// Mitsubishi GX Developer project: PLC_PCO520L2   PLC: Q06UDEH

PROGRAM MAIN
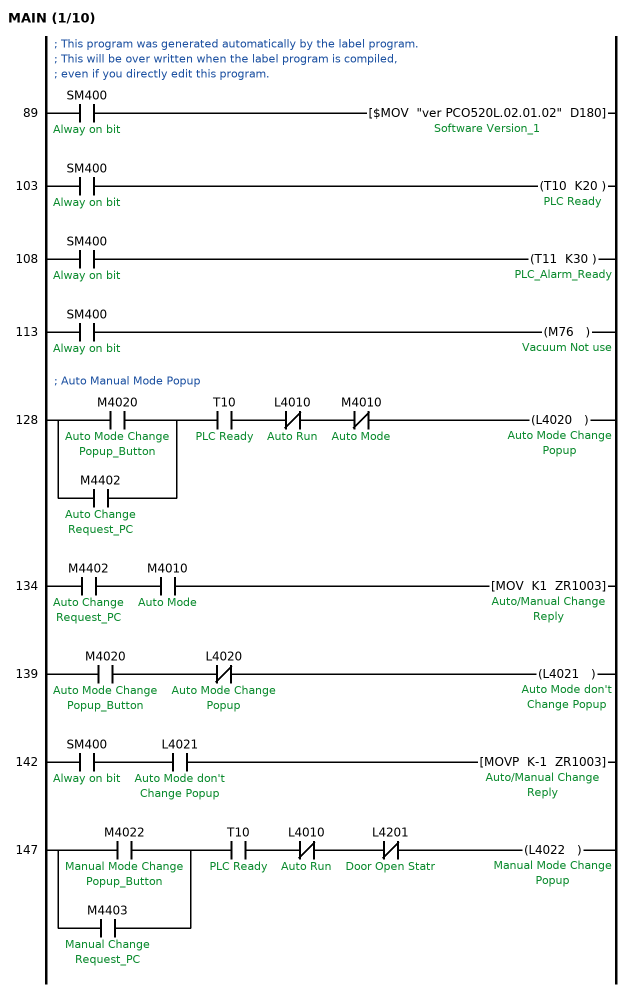
; This program was generated automatically by the label program.
; This will be over written when the label program is compiled,
; even if you directly edit this program.
89    LD      SM400  ; Alway on bit
      $MOV    "ver PCO520L.02.01.02" D180  ; Software Version_1
103   LD      SM400  ; Alway on bit
      OUT     T10 K20  ; PLC Ready
108   LD      SM400  ; Alway on bit
      OUT     T11 K30  ; PLC_Alarm_Ready
113   LD      SM400  ; Alway on bit
      OUT     M76  ; Vacuum Not use
; Auto Manual Mode Popup
128   LD      M4020  ; Auto Mode Change Popup_Button
      OR      M4402  ; Auto Change Request_PC
      AND     T10  ; PLC Ready
      ANI     L4010  ; Auto Run
      ANI     M4010  ; Auto Mode
      OUT     L4020  ; Auto Mode Change Popup
134   LD      M4402  ; Auto Change Request_PC
      AND     M4010  ; Auto Mode
      MOV     K1 ZR1003  ; Auto/Manual Change Reply
139   LD      M4020  ; Auto Mode Change Popup_Button
      ANI     L4020  ; Auto Mode Change Popup
      OUT     L4021  ; Auto Mode don't Change Popup
142   LD      SM400  ; Alway on bit
      AND     L4021  ; Auto Mode don't Change Popup
      MOVP    K-1 ZR1003
147   LD      M4022  ; Manual Mode Change Popup_Button
      OR      M4403  ; Manual Change Request_PC
      AND     T10  ; PLC Ready
      ANI     L4010  ; Auto Run
      ANI     L4201  ; Door Open Statr
      OUT     L4022  ; Manual Mode Change Popup
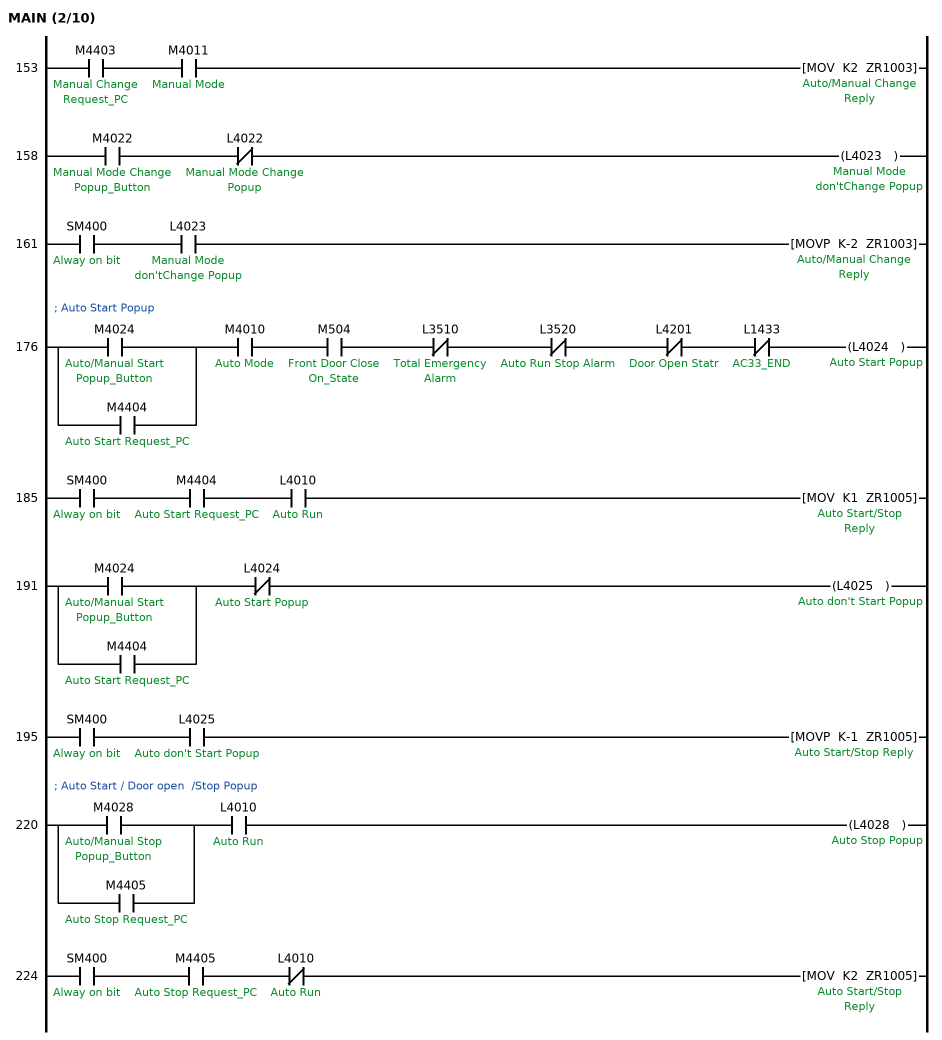
153   LD      M4403  ; Manual Change Request_PC
      AND     M4011  ; Manual Mode
      MOV     K2 ZR1003
158   LD      M4022  ; Manual Mode Change Popup_Button
      ANI     L4022  ; Manual Mode Change Popup
      OUT     L4023  ; Manual Mode  don'tChange Popup
161   LD      SM400  ; Alway on bit
      AND     L4023  ; Manual Mode  don'tChange Popup
      MOVP    K-2 ZR1003
; Auto Start Popup
176   LD      M4024  ; Auto/Manual Start Popup_Button
      OR      M4404  ; Auto Start Request_PC
      AND     M4010  ; Auto Mode
      AND     M504  ; Front Door Close On_State
      ANI     L3510  ; Total Emergency Alarm
      ANI     L3520  ; Auto Run Stop Alarm
      ANI     L4201  ; Door Open Statr
      ANI     L1433  ; AC33_END
      OUT     L4024  ; Auto Start Popup
185   LD      SM400  ; Alway on bit
      AND     M4404  ; Auto Start Request_PC
      AND     L4010  ; Auto Run
      MOV     K1 ZR1005  ; Auto Start/Stop Reply
191   LD      M4024  ; Auto/Manual Start Popup_Button
      OR      M4404  ; Auto Start Request_PC
      ANI     L4024  ; Auto Start Popup
      OUT     L4025  ; Auto don't Start Popup
195   LD      SM400  ; Alway on bit
      AND     L4025  ; Auto don't Start Popup
      MOVP    K-1 ZR1005
; Auto Start / Door open  /Stop Popup
220   LD      M4028  ; Auto/Manual Stop Popup_Button
      OR      M4405  ; Auto Stop Request_PC
      AND     L4010  ; Auto Run
      OUT     L4028  ; Auto Stop Popup
224   LD      SM400  ; Alway on bit
      AND     M4405  ; Auto Stop Request_PC
      ANI     L4010  ; Auto Run
      MOV     K2 ZR1005
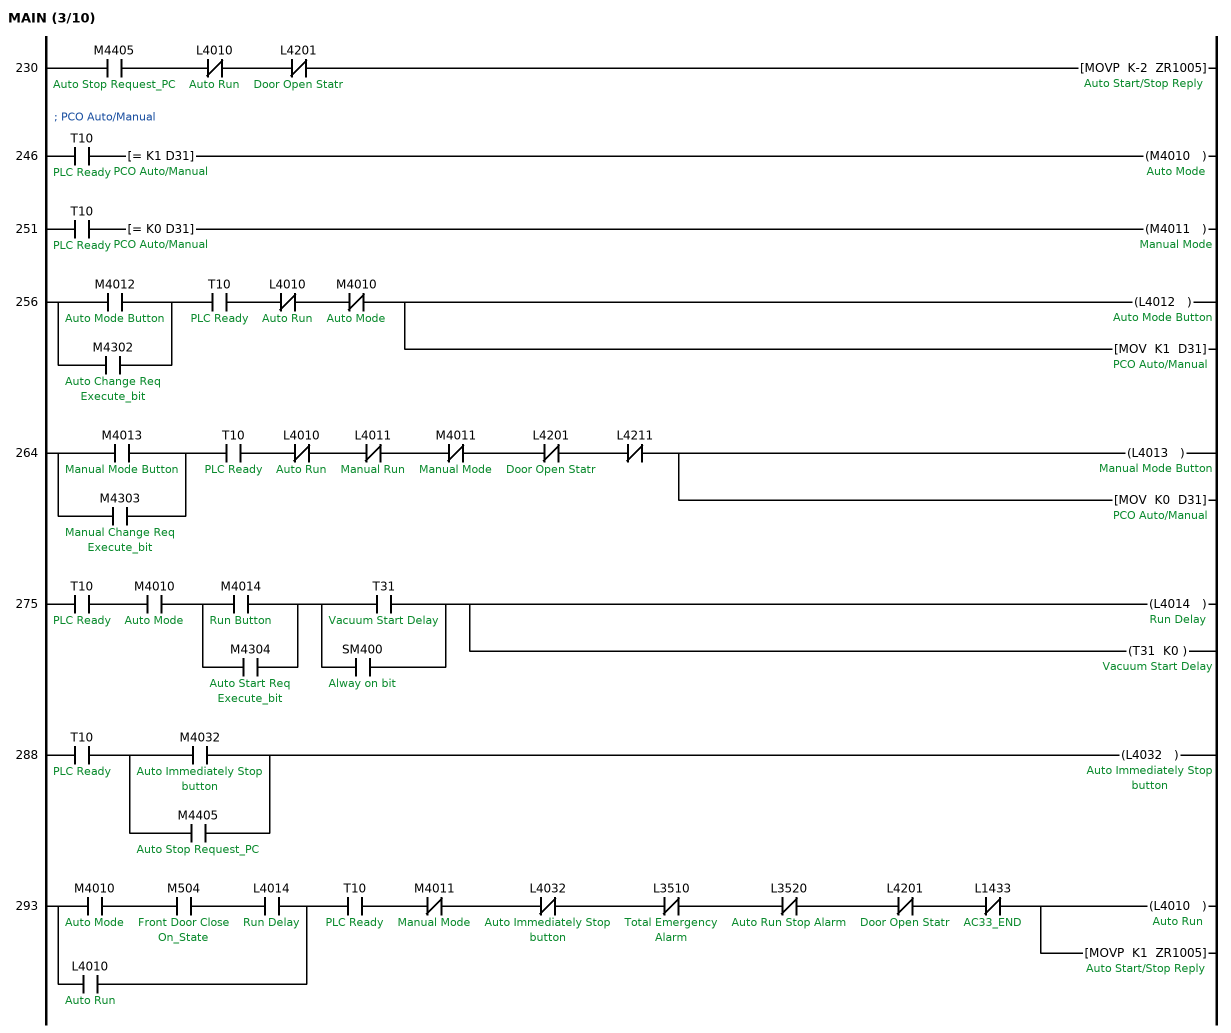
230   LD      M4405  ; Auto Stop Request_PC
      ANI     L4010  ; Auto Run
      ANI     L4201  ; Door Open Statr
      MOVP    K-2 ZR1005
; PCO Auto/Manual
246   LD      T10  ; PLC Ready
      AND=    K1 D31  ; PCO Auto/Manual
      OUT     M4010  ; Auto Mode
251   LD      T10  ; PLC Ready
      AND=    K0 D31  ; PCO Auto/Manual
      OUT     M4011  ; Manual Mode
256   LD      M4012  ; Auto Mode Button
      OR      M4302  ; Auto Change Req Execute_bit
      AND     T10  ; PLC Ready
      ANI     L4010  ; Auto Run
      ANI     M4010  ; Auto Mode
      OUT     L4012  ; Auto Mode Button
      MOV     K1 D31
264   LD      M4013  ; Manual Mode Button
      OR      M4303  ; Manual Change Req Execute_bit
      AND     T10  ; PLC Ready
      ANI     L4010  ; Auto Run
      ANI     L4011  ; Manual Run
      ANI     M4011  ; Manual Mode
      ANI     L4201  ; Door Open Statr
      ANI     L4211
      OUT     L4013  ; Manual Mode Button
      MOV     K0 D31
275   LD      T10  ; PLC Ready
      AND     M4010  ; Auto Mode
      LD      M4014  ; Run Button
      OR      M4304  ; Auto Start Req Execute_bit
      ANB
      LD      T31  ; Vacuum Start Delay
      OR      SM400  ; Alway on bit
      ANB
      OUT     L4014  ; Run Delay
      OUT     T31 K0  ; Vacuum Start Delay
288   LD      T10  ; PLC Ready
      LD      M4032  ; Auto Immediately Stop button
      OR      M4405  ; Auto Stop Request_PC
      ANB
      OUT     L4032  ; Auto Immediately Stop button
293   LD      M4010  ; Auto Mode
      AND     M504  ; Front Door Close On_State
      AND     L4014  ; Run Delay
      OR      L4010  ; Auto Run
      AND     T10  ; PLC Ready
      ANI     M4011  ; Manual Mode
      ANI     L4032  ; Auto Immediately Stop button
      ANI     L3510  ; Total Emergency Alarm
      ANI     L3520  ; Auto Run Stop Alarm
      ANI     L4201  ; Door Open Statr
      ANI     L1433  ; AC33_END
      OUT     L4010  ; Auto Run
      MOVP    K1 ZR1005
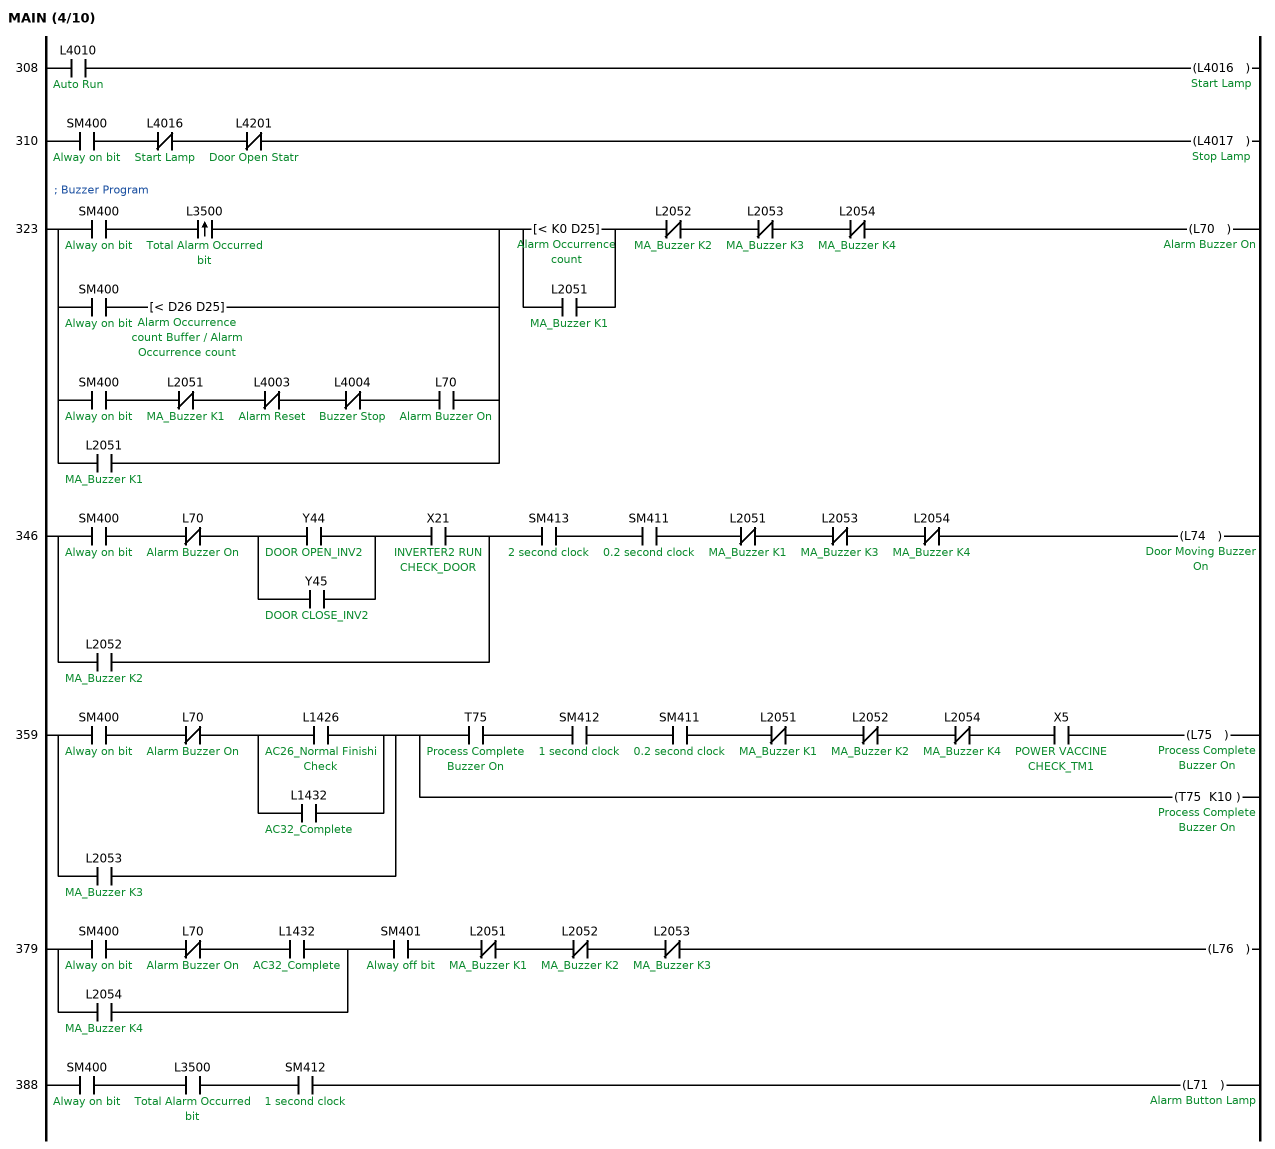
308   LD      L4010  ; Auto Run
      OUT     L4016  ; Start Lamp
310   LD      SM400  ; Alway on bit
      ANI     L4016  ; Start Lamp
      ANI     L4201  ; Door Open Statr
      OUT     L4017  ; Stop Lamp
; Buzzer Program
323   LD      SM400  ; Alway on bit
      ANDP    L3500  ; Total Alarm Occurred bit
      LD      SM400  ; Alway on bit
      AND<    D26 D25  ; Alarm Occurrence count Buffer / Alarm Occurrence count
      ORB
      LD      SM400  ; Alway on bit
      ANI     L2051  ; MA_Buzzer K1
      ANI     L4003  ; Alarm Reset
      ANI     L4004  ; Buzzer Stop
      AND     L70  ; Alarm Buzzer On
      ORB
      OR      L2051  ; MA_Buzzer K1
      LD<     K0 D25  ; Alarm Occurrence count
      OR      L2051  ; MA_Buzzer K1
      ANB
      ANI     L2052  ; MA_Buzzer K2
      ANI     L2053  ; MA_Buzzer K3
      ANI     L2054  ; MA_Buzzer K4
      OUT     L70  ; Alarm Buzzer On
346   LD      SM400  ; Alway on bit
      ANI     L70  ; Alarm Buzzer On
      LD      Y44  ; DOOR OPEN_INV2
      OR      Y45  ; DOOR CLOSE_INV2
      ANB
      AND     X21  ; INVERTER2 RUN CHECK_DOOR
      OR      L2052  ; MA_Buzzer K2
      AND     SM413  ; 2 second clock
      AND     SM411  ; 0.2 second clock
      ANI     L2051  ; MA_Buzzer K1
      ANI     L2053  ; MA_Buzzer K3
      ANI     L2054  ; MA_Buzzer K4
      OUT     L74  ; Door Moving Buzzer On
359   LD      SM400  ; Alway on bit
      ANI     L70  ; Alarm Buzzer On
      LD      L1426  ; AC26_Normal Finishi Check
      OR      L1432  ; AC32_Complete
      ANB
      OR      L2053  ; MA_Buzzer K3
      MPS
      AND     T75  ; Process Complete Buzzer On
      AND     SM412  ; 1 second clock
      AND     SM411  ; 0.2 second clock
      ANI     L2051  ; MA_Buzzer K1
      ANI     L2052  ; MA_Buzzer K2
      ANI     L2054  ; MA_Buzzer K4
      AND     X5  ; POWER VACCINE CHECK_TM1
      OUT     L75  ; Process Complete Buzzer On
      MPP
      OUT     T75 K10  ; Process Complete Buzzer On
379   LD      SM400  ; Alway on bit
      ANI     L70  ; Alarm Buzzer On
      AND     L1432  ; AC32_Complete
      OR      L2054  ; MA_Buzzer K4
      AND     SM401  ; Alway off bit
      ANI     L2051  ; MA_Buzzer K1
      ANI     L2052  ; MA_Buzzer K2
      ANI     L2053  ; MA_Buzzer K3
      OUT     L76
388   LD      SM400  ; Alway on bit
      AND     L3500  ; Total Alarm Occurred bit
      AND     SM412  ; 1 second clock
      OUT     L71  ; Alarm Button Lamp
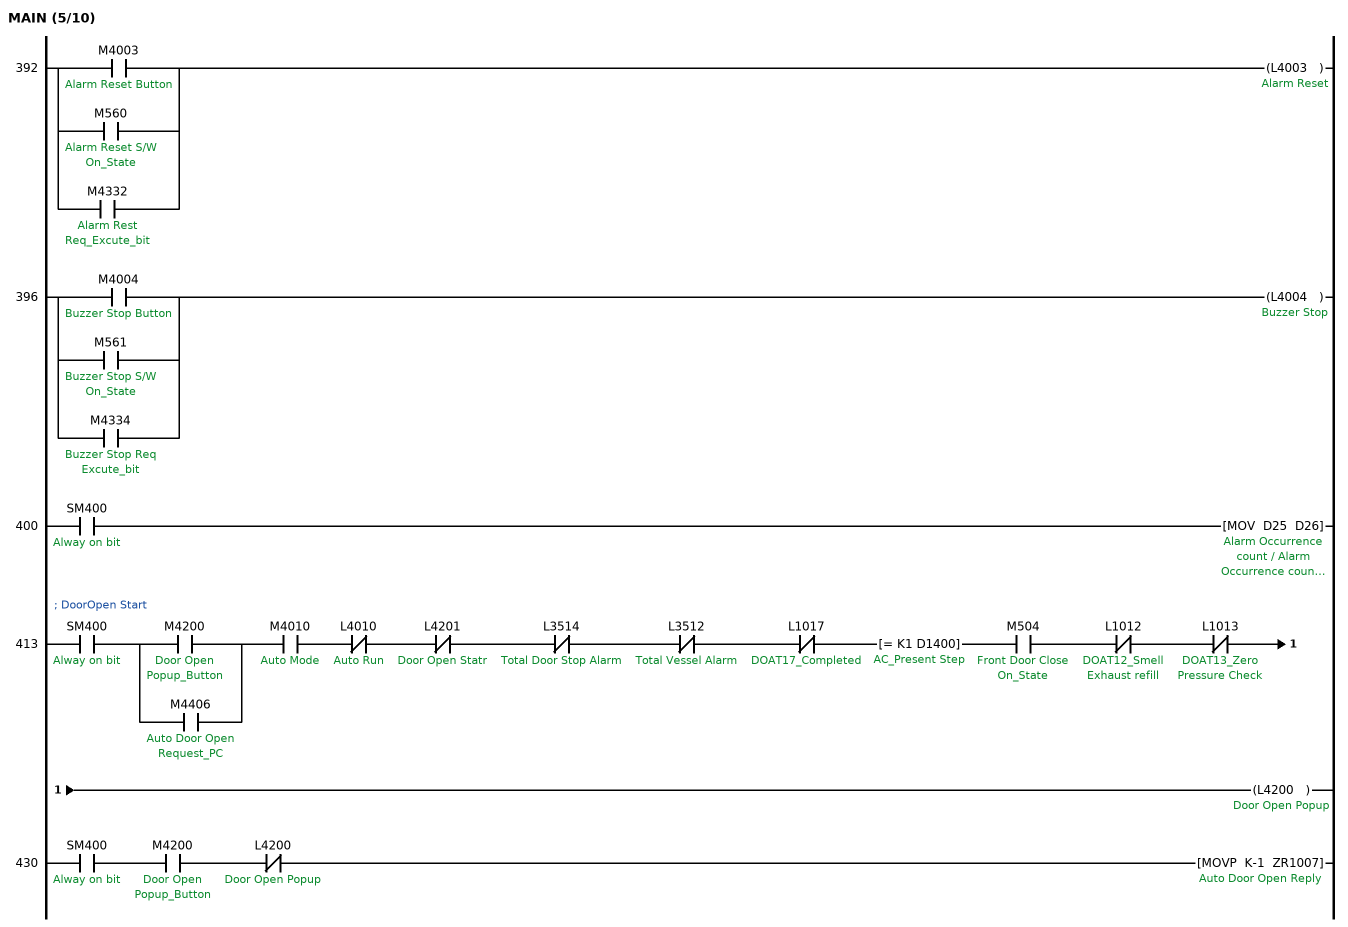
392   LD      M4003  ; Alarm Reset Button
      OR      M560  ; Alarm Reset S/W On_State
      OR      M4332  ; Alarm Rest Req_Excute_bit
      OUT     L4003  ; Alarm Reset
396   LD      M4004  ; Buzzer Stop Button
      OR      M561  ; Buzzer Stop S/W On_State
      OR      M4334  ; Buzzer Stop Req Excute_bit
      OUT     L4004  ; Buzzer Stop
400   LD      SM400  ; Alway on bit
      MOV     D25 D26
; DoorOpen Start
413   LD      SM400  ; Alway on bit
      LD      M4200  ; Door Open Popup_Button
      OR      M4406  ; Auto Door Open Request_PC
      ANB
      AND     M4010  ; Auto Mode
      ANI     L4010  ; Auto Run
      ANI     L4201  ; Door Open Statr
      ANI     L3514  ; Total Door Stop Alarm
      ANI     L3512  ; Total Vessel Alarm
      ANI     L1017  ; DOAT17_Completed
      AND=    K1 D1400  ; AC_Present Step
      AND     M504  ; Front Door Close On_State
      ANI     L1012  ; DOAT12_Smell Exhaust refill
      ANI     L1013  ; DOAT13_Zero Pressure Check
      OUT     L4200  ; Door Open Popup
430   LD      SM400  ; Alway on bit
      AND     M4200  ; Door Open Popup_Button
      ANI     L4200  ; Door Open Popup
      MOVP    K-1 ZR1007  ; Auto Door Open Reply
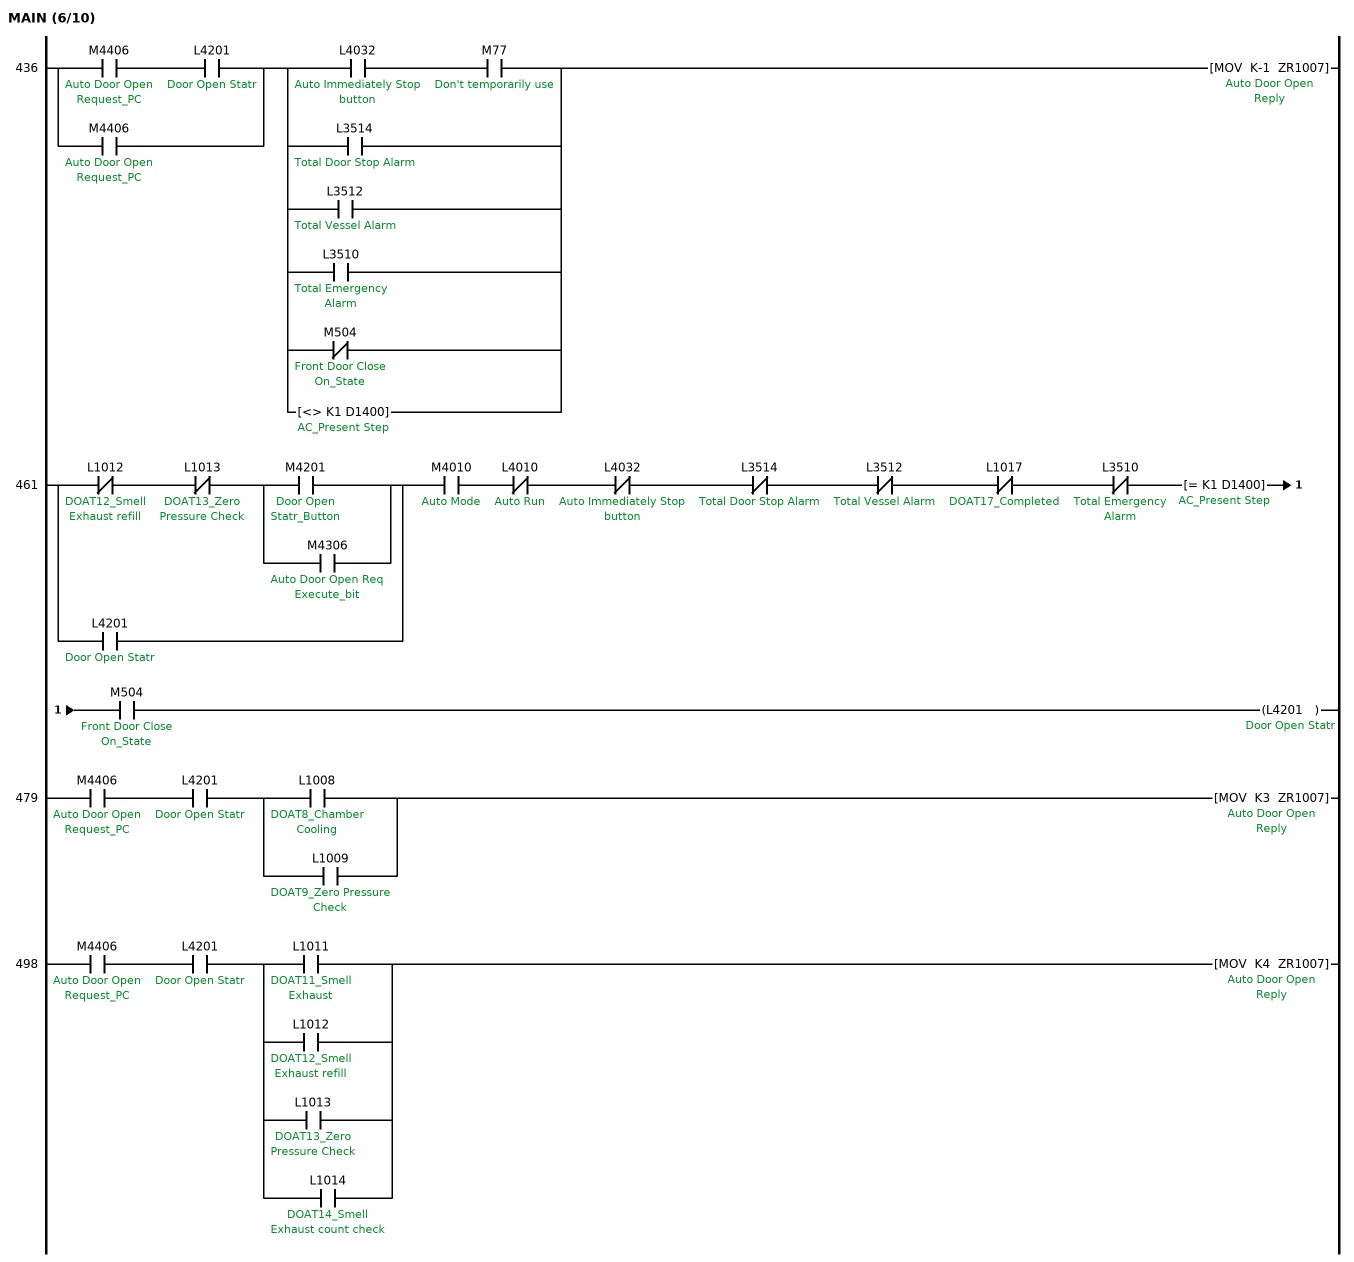
436   LD      M4406  ; Auto Door Open Request_PC
      AND     L4201  ; Door Open Statr
      OR      M4406  ; Auto Door Open Request_PC
      LD      L4032  ; Auto Immediately Stop button
      AND     M77  ; Don't temporarily use
      OR      L3514  ; Total Door Stop Alarm
      OR      L3512  ; Total Vessel Alarm
      OR      L3510  ; Total Emergency Alarm
      ORI     M504  ; Front Door Close On_State
      OR<>    K1 D1400  ; AC_Present Step
      ANB
      MOV     K-1 ZR1007
        [note] Door Open fail
461   LDI     L1012  ; DOAT12_Smell Exhaust refill
      ANI     L1013  ; DOAT13_Zero Pressure Check
      LD      M4201  ; Door Open Statr_Button
      OR      M4306  ; Auto Door Open Req Execute_bit
      ANB
      OR      L4201  ; Door Open Statr
      AND     M4010  ; Auto Mode
      ANI     L4010  ; Auto Run
      ANI     L4032  ; Auto Immediately Stop button
      ANI     L3514  ; Total Door Stop Alarm
      ANI     L3512  ; Total Vessel Alarm
      ANI     L1017  ; DOAT17_Completed
      ANI     L3510  ; Total Emergency Alarm
      AND=    K1 D1400  ; AC_Present Step
      AND     M504  ; Front Door Close On_State
      OUT     L4201  ; Door Open Statr
479   LD      M4406  ; Auto Door Open Request_PC
      AND     L4201  ; Door Open Statr
      LD      L1008  ; DOAT8_Chamber Cooling
      OR      L1009  ; DOAT9_Zero Pressure Check
      ANB
      MOV     K3 ZR1007
        [note] Cooling Inprogress
498   LD      M4406  ; Auto Door Open Request_PC
      AND     L4201  ; Door Open Statr
      LD      L1011  ; DOAT11_Smell Exhaust
      OR      L1012  ; DOAT12_Smell Exhaust refill
      OR      L1013  ; DOAT13_Zero Pressure Check
      OR      L1014  ; DOAT14_Smell Exhaust count check
      ANB
      MOV     K4 ZR1007
        [note] Smell Exhaust Inprogress
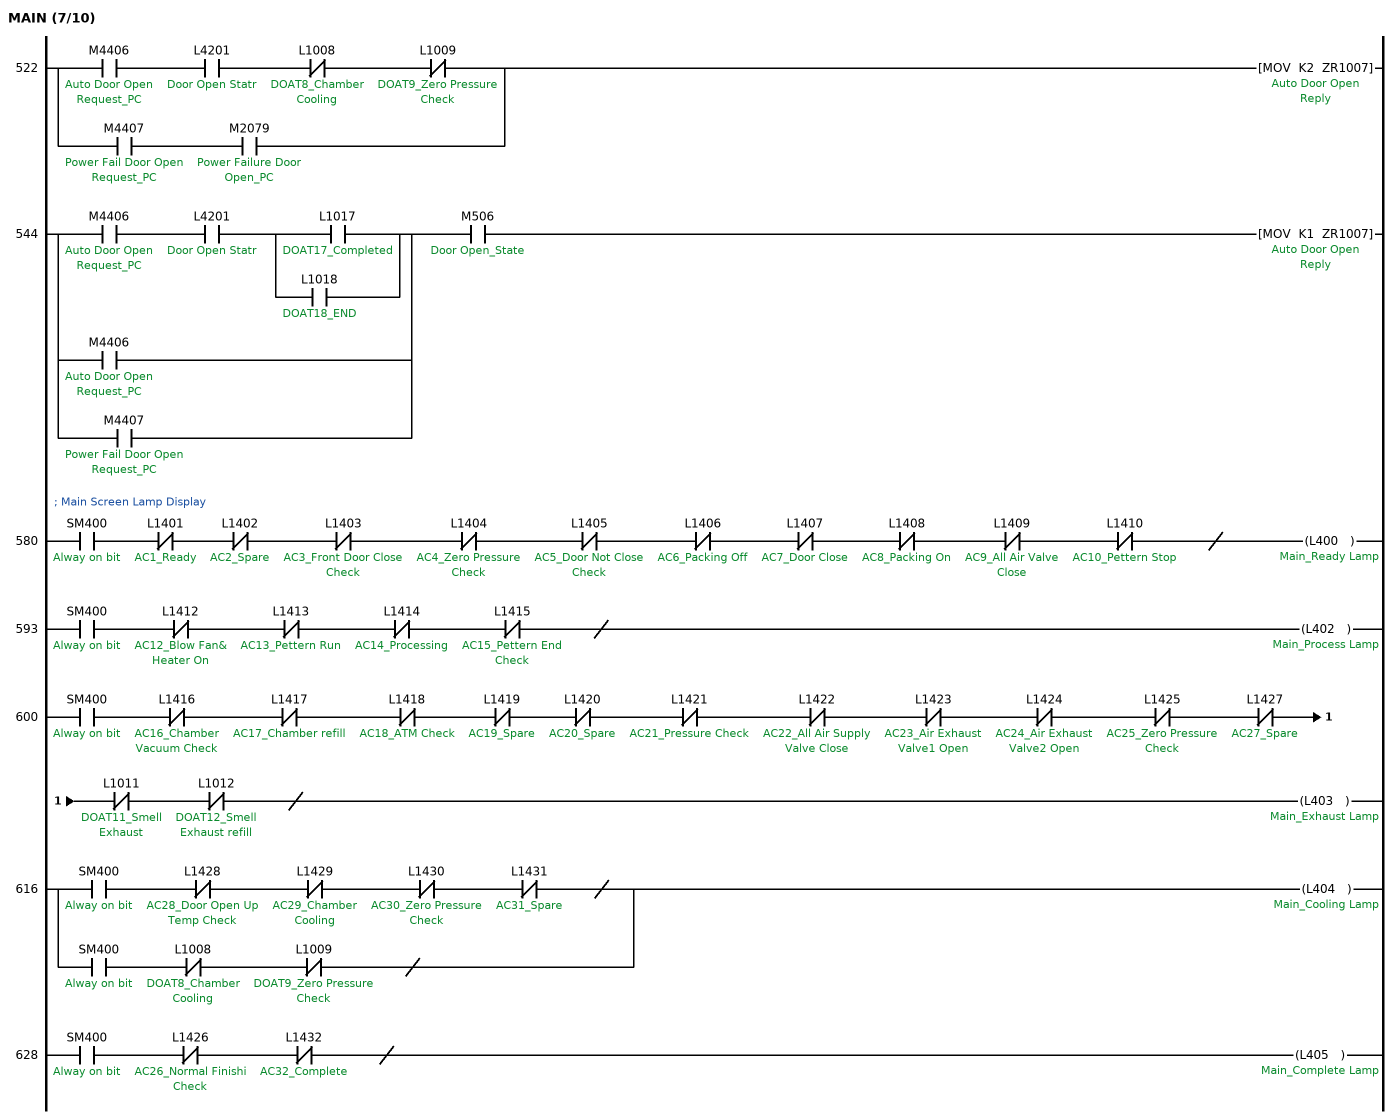
522   LD      M4406  ; Auto Door Open Request_PC
      AND     L4201  ; Door Open Statr
      ANI     L1008  ; DOAT8_Chamber Cooling
      ANI     L1009  ; DOAT9_Zero Pressure Check
      LD      M4407  ; Power Fail Door Open Request_PC
      AND     M2079  ; Power Failure Door Open_PC
      ORB
      MOV     K2 ZR1007
        [note] Door Open Inprogress
544   LD      M4406  ; Auto Door Open Request_PC
      AND     L4201  ; Door Open Statr
      LD      L1017  ; DOAT17_Completed
      OR      L1018  ; DOAT18_END
      ANB
      OR      M4406  ; Auto Door Open Request_PC
      OR      M4407  ; Power Fail Door Open Request_PC
      AND     M506  ; Door Open_State
      MOV     K1 ZR1007
        [note] Door Open Complete
; Main Screen Lamp Display
580   LD      SM400  ; Alway on bit
      ANI     L1401  ; AC1_Ready
      ANI     L1402  ; AC2_Spare
      ANI     L1403  ; AC3_Front Door Close Check
      ANI     L1404  ; AC4_Zero Pressure Check
      ANI     L1405  ; AC5_Door Not Close Check
      ANI     L1406  ; AC6_Packing Off
      ANI     L1407  ; AC7_Door Close
      ANI     L1408  ; AC8_Packing On
      ANI     L1409  ; AC9_All Air Valve Close
      ANI     L1410  ; AC10_Pettern Stop
      INV
      OUT     L400  ; Main_Ready Lamp
593   LD      SM400  ; Alway on bit
      ANI     L1412  ; AC12_Blow Fan& Heater On
      ANI     L1413  ; AC13_Pettern Run
      ANI     L1414  ; AC14_Processing
      ANI     L1415  ; AC15_Pettern End Check
      INV
      OUT     L402  ; Main_Process Lamp
600   LD      SM400  ; Alway on bit
      ANI     L1416  ; AC16_Chamber Vacuum Check
      ANI     L1417  ; AC17_Chamber refill
      ANI     L1418  ; AC18_ATM Check
      ANI     L1419  ; AC19_Spare
      ANI     L1420  ; AC20_Spare
      ANI     L1421  ; AC21_Pressure Check
      ANI     L1422  ; AC22_All Air Supply Valve Close
      ANI     L1423  ; AC23_Air Exhaust Valve1 Open
      ANI     L1424  ; AC24_Air Exhaust Valve2 Open
      ANI     L1425  ; AC25_Zero Pressure Check
      ANI     L1427  ; AC27_Spare
      ANI     L1011  ; DOAT11_Smell Exhaust
      ANI     L1012  ; DOAT12_Smell Exhaust refill
      INV
      OUT     L403  ; Main_Exhaust Lamp
616   LD      SM400  ; Alway on bit
      ANI     L1428  ; AC28_Door Open Up Temp Check
      ANI     L1429  ; AC29_Chamber Cooling
      ANI     L1430  ; AC30_Zero Pressure Check
      ANI     L1431  ; AC31_Spare
      INV
      LD      SM400  ; Alway on bit
      ANI     L1008  ; DOAT8_Chamber Cooling
      ANI     L1009  ; DOAT9_Zero Pressure Check
      INV
      ORB
      OUT     L404  ; Main_Cooling Lamp
628   LD      SM400  ; Alway on bit
      ANI     L1426  ; AC26_Normal Finishi Check
      ANI     L1432  ; AC32_Complete
      INV
      OUT     L405  ; Main_Complete Lamp
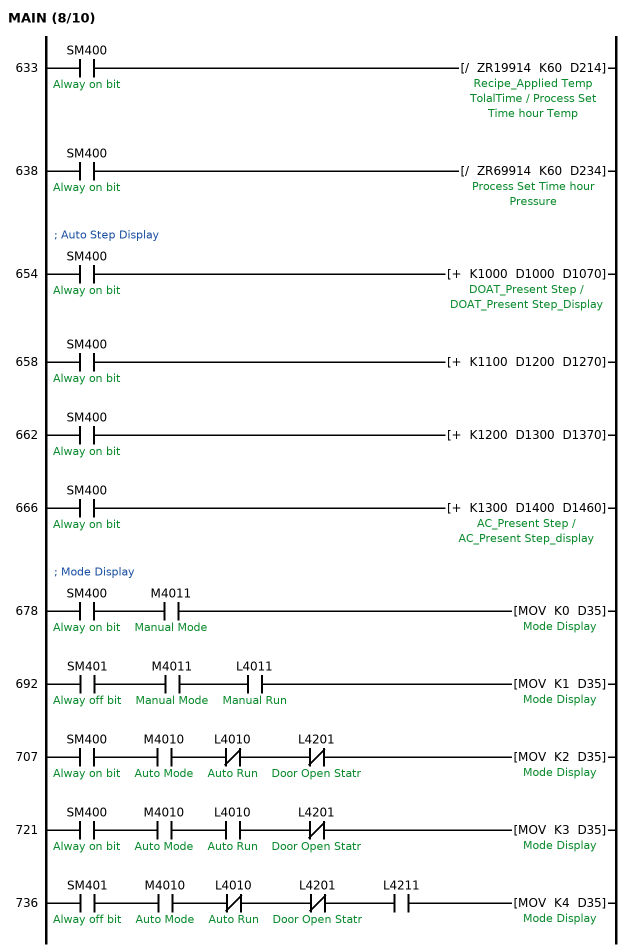
633   LD      SM400  ; Alway on bit
      /       ZR19914 K60 D214  ; Recipe_Applied Temp TolalTime / Process Set Time hour Temp
638   LD      SM400  ; Alway on bit
      /       ZR69914 K60 D234  ; Process Set Time hour Pressure
; Auto Step Display
654   LD      SM400  ; Alway on bit
      +       K1000 D1000 D1070  ; DOAT_Present Step / DOAT_Present Step_Display
658   LD      SM400  ; Alway on bit
      +       K1100 D1200 D1270
662   LD      SM400  ; Alway on bit
      +       K1200 D1300 D1370
666   LD      SM400  ; Alway on bit
      +       K1300 D1400 D1460  ; AC_Present Step_display
; Mode Display
678   LD      SM400  ; Alway on bit
      AND     M4011  ; Manual Mode
      MOV     K0 D35  ; Mode Display
        [note] 0: Manual Mode
692   LD      SM401  ; Alway off bit
      AND     M4011  ; Manual Mode
      AND     L4011  ; Manual Run
      MOV     K1 D35
        [note] 1: Manual Start
707   LD      SM400  ; Alway on bit
      AND     M4010  ; Auto Mode
      ANI     L4010  ; Auto Run
      ANI     L4201  ; Door Open Statr
      MOV     K2 D35
        [note] 2: Auto Mode
721   LD      SM400  ; Alway on bit
      AND     M4010  ; Auto Mode
      AND     L4010  ; Auto Run
      ANI     L4201  ; Door Open Statr
      MOV     K3 D35
        [note] 3: Auto Start
736   LD      SM401  ; Alway off bit
      AND     M4010  ; Auto Mode
      ANI     L4010  ; Auto Run
      ANI     L4201  ; Door Open Statr
      AND     L4211
      MOV     K4 D35
        [note] Preheat Start
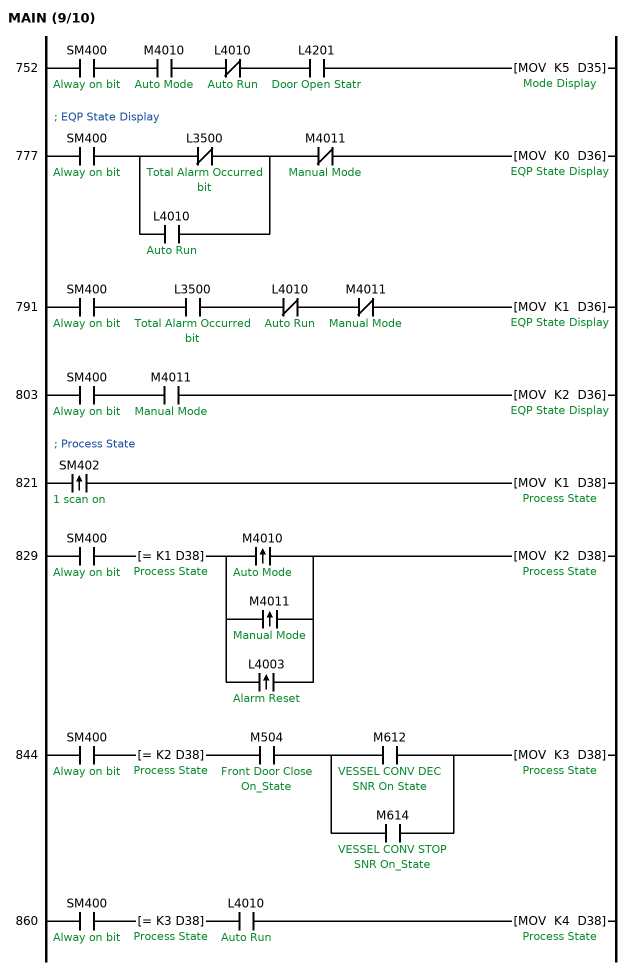
752   LD      SM400  ; Alway on bit
      AND     M4010  ; Auto Mode
      ANI     L4010  ; Auto Run
      AND     L4201  ; Door Open Statr
      MOV     K5 D35
        [note] 5: Door Open
; EQP State Display
777   LD      SM400  ; Alway on bit
      LDI     L3500  ; Total Alarm Occurred bit
      OR      L4010  ; Auto Run
      ANB
      ANI     M4011  ; Manual Mode
      MOV     K0 D36  ; EQP State Display
        [note] 0: Normal
791   LD      SM400  ; Alway on bit
      AND     L3500  ; Total Alarm Occurred bit
      ANI     L4010  ; Auto Run
      ANI     M4011  ; Manual Mode
      MOV     K1 D36
        [note] 1: Fault
803   LD      SM400  ; Alway on bit
      AND     M4011  ; Manual Mode
      MOV     K2 D36
        [note] 2: PM
; Process State
821   LDP     SM402  ; 1 scan on
      MOV     K1 D38  ; Process State
        [note] 1: INT
829   LD      SM400  ; Alway on bit
      AND=    K1 D38  ; Process State
      LDP     M4010  ; Auto Mode
      ORP     M4011  ; Manual Mode
      ORP     L4003  ; Alarm Reset
      ANB
      MOV     K2 D38
        [note] 2:LOAD
844   LD      SM400  ; Alway on bit
      AND=    K2 D38  ; Process State
      AND     M504  ; Front Door Close On_State
      LD      M612  ; VESSEL CONV DEC SNR On State
      OR      M614  ; VESSEL CONV STOP SNR On_State
      ANB
      MOV     K3 D38
        [note] 3:READY
860   LD      SM400  ; Alway on bit
      AND=    K3 D38  ; Process State
      AND     L4010  ; Auto Run
      MOV     K4 D38
        [note] 4:EXECUTING
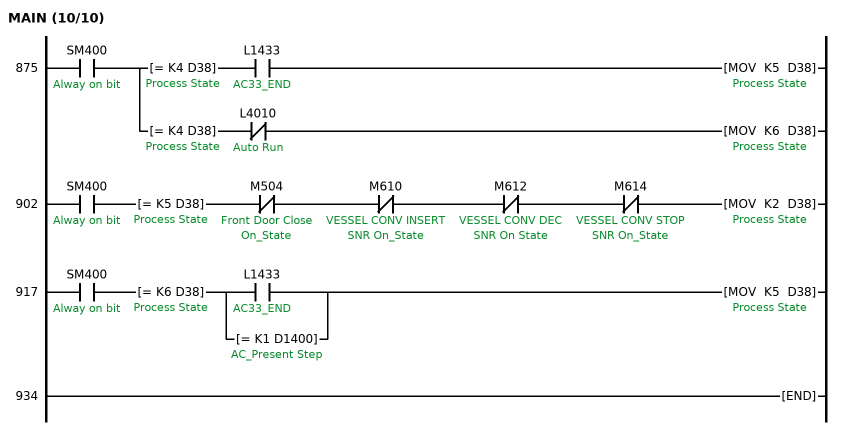
875   LD      SM400  ; Alway on bit
      MPS
      AND=    K4 D38  ; Process State
      AND     L1433  ; AC33_END
      MOV     K5 D38
        [note] 5:UNLOAD
      MPP
      AND=    K4 D38  ; Process State
      ANI     L4010  ; Auto Run
      MOV     K6 D38
        [note] 6:ABORT
902   LD      SM400  ; Alway on bit
      AND=    K5 D38  ; Process State
      ANI     M504  ; Front Door Close On_State
      ANI     M610  ; VESSEL CONV INSERT SNR On_State
      ANI     M612  ; VESSEL CONV DEC SNR On State
      ANI     M614  ; VESSEL CONV STOP SNR On_State
      MOV     K2 D38
        [note] 2:LOAD
917   LD      SM400  ; Alway on bit
      AND=    K6 D38  ; Process State
      LD      L1433  ; AC33_END
      OR=     K1 D1400  ; AC_Present Step
      ANB
      MOV     K5 D38
        [note] 5:UNLOAD
934   END
END_PROGRAM
